FUNCTION_BLOCK FB_Pump
VAR_INPUT
END_VAR
VAR_OUTPUT
END_VAR
VAR
	
 // For logging
    fbLogger : FB_LogMessage := (eSubsystem:=E_SubSystem.VACUUM);
    ePrevState : E_PumpState;
    tErrorPresent : R_TRIG;
    tAction : R_TRIG; // Primary action of this device (OPN_DO, PUMP_RUN, etc.)	
	tFault : F_TRIG;
	tILK: TON;
END_VAR

ACTION ACT_Logger:

END_ACTION

END_FUNCTION_BLOCK

(* stored: Version 1.1.0.1, ProductVersion 3.1.4022.18
   POU FB_Pump: Id {00c4f02d-0992-44f0-9021-57d8126c2097}, SpecialFunc None
   Action ACT_Logger: Id {3638f3f4-c294-44fa-a1a7-c4bfc15b56a5} *)
